// TIA Portal V19 export
ORGANIZATION_BLOCK "Main_hw"   // OB124, LAD, ProgramCycle
TITLE = "Main Program Sweep (Cycle)"
{ S7_Optimized_Access := 'TRUE' }
// stored: SetENOAutomatically false
   VAR_INPUT
      Initial_Call : Bool;   // Initial call of this OB
      Remanence : Bool;   // =True, if remanent data are available
   END_VAR
   VAR_TEMP   // added for the SCL form of the ladder/FBD networks
      _w1 : Bool;
      _w2 : Bool;
   END_VAR
BEGIN

REGION Network 1: HMI hardware test screen control
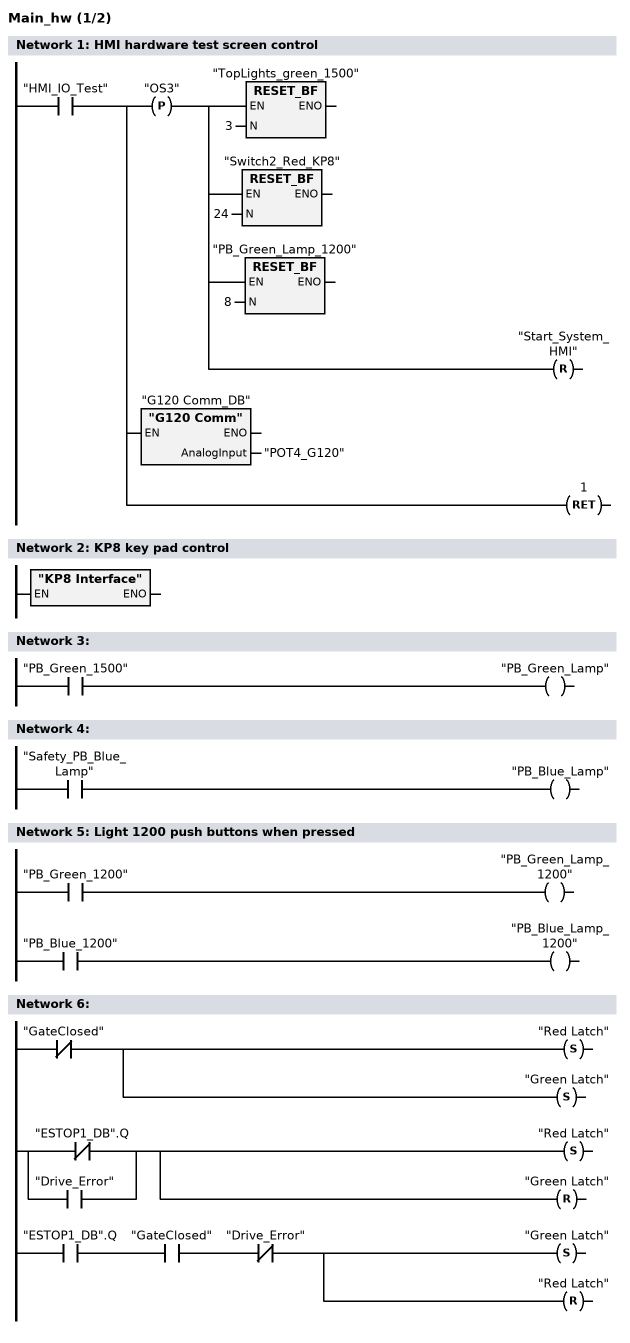
   // no SCL statement known for RBitfield: written as a call
   #_w1 := "HMI_IO_Test" AND NOT "OS3";   // rising edge
   "OS3" := "HMI_IO_Test";
   #_w2 := "HMI_IO_Test";
   IF #_w1 THEN
       RESET_BF(operand := "TopLights_green_1500", n := 3);
       RESET_BF(operand := "Switch2_Red_KP8", n := 24);
       RESET_BF(operand := "PB_Green_Lamp_1200", n := 8);
       "Start_System_HMI" := FALSE;
   END_IF;
   IF #_w2 THEN
       "G120 Comm_DB"(AnalogInput => "POT4_G120");   // "G120 Comm"
       ENO := 1;
       RETURN;
   END_IF;
END_REGION

REGION Network 2: KP8 key pad control
   RUNG wire#powerrail
      "KP8 Interface"()
   END_RUNG
   // the same network as SCL:
   "KP8 Interface"();
END_REGION

REGION Network 3
   RUNG wire#powerrail
      Contact( "PB_Green_1500" )
      Coil( "PB_Green_Lamp" )
   END_RUNG
   // the same network as SCL:
   "PB_Green_Lamp" := "PB_Green_1500";
END_REGION

REGION Network 4
   RUNG wire#powerrail
      Contact( "Safety_PB_Blue_Lamp" )
      Coil( "PB_Blue_Lamp" )
   END_RUNG
   // the same network as SCL:
   "PB_Blue_Lamp" := "Safety_PB_Blue_Lamp";
END_REGION

REGION Network 5: Light 1200 push buttons when pressed
   RUNG wire#powerrail
      Contact( "PB_Green_1200" )
      Coil( "PB_Green_Lamp_1200" )
   END_RUNG
   RUNG wire#powerrail
      Contact( "PB_Blue_1200" )
      Coil( "PB_Blue_Lamp_1200" )
   END_RUNG
   // the same network as SCL:
   "PB_Green_Lamp_1200" := "PB_Green_1200";
   "PB_Blue_Lamp_1200" := "PB_Blue_1200";
END_REGION

REGION Network 6
   RUNG wire#powerrail
      I_Contact( "GateClosed" )
      wire#w1
      S_Coil( "Red Latch" )
   END_RUNG
   RUNG wire#w1
      S_Coil( "Green Latch" )
   END_RUNG
   RUNG wire#powerrail
      I_Contact( "ESTOP1_DB".Q )
      wire#w2
      S_Coil( "Red Latch" )
   END_RUNG
   RUNG wire#powerrail
      Contact( "Drive_Error" )
   END_RUNG wire#w2
   RUNG wire#w2
      R_Coil( "Green Latch" )
   END_RUNG
   RUNG wire#powerrail
      Contact( "ESTOP1_DB".Q )
      Contact( "GateClosed" )
      I_Contact( "Drive_Error" )
      wire#w3
      S_Coil( "Green Latch" )
   END_RUNG
   RUNG wire#w3
      R_Coil( "Red Latch" )
   END_RUNG
   // the same network as SCL:
   IF NOT "GateClosed" THEN
       "Red Latch" := TRUE;
       "Green Latch" := TRUE;
   END_IF;
   IF NOT "ESTOP1_DB".Q OR "Drive_Error" THEN
       "Red Latch" := TRUE;
       "Green Latch" := FALSE;
   END_IF;
   IF "ESTOP1_DB".Q AND "GateClosed" AND NOT "Drive_Error" THEN
       "Green Latch" := TRUE;
       "Red Latch" := FALSE;
   END_IF;
END_REGION

REGION Network 7
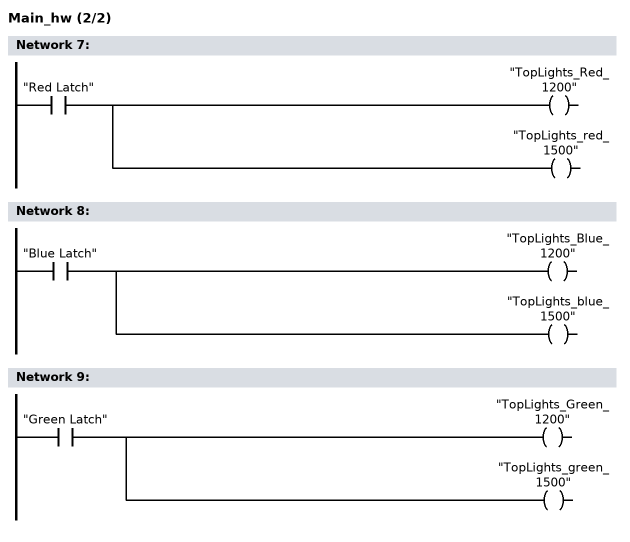
   RUNG wire#powerrail
      Contact( "Red Latch" )
      wire#w1
      Coil( "TopLights_Red_1200" )
   END_RUNG
   RUNG wire#w1
      Coil( "TopLights_red_1500" )
   END_RUNG
   // the same network as SCL:
   "TopLights_Red_1200" := "Red Latch";
   "TopLights_red_1500" := "Red Latch";
END_REGION

REGION Network 8
   RUNG wire#powerrail
      Contact( "Blue Latch" )
      wire#w1
      Coil( "TopLights_Blue_1200" )
   END_RUNG
   RUNG wire#w1
      Coil( "TopLights_blue_1500" )
   END_RUNG
   // the same network as SCL:
   "TopLights_Blue_1200" := "Blue Latch";
   "TopLights_blue_1500" := "Blue Latch";
END_REGION

REGION Network 9
   RUNG wire#powerrail
      Contact( "Green Latch" )
      wire#w1
      Coil( "TopLights_Green_1200" )
   END_RUNG
   RUNG wire#w1
      Coil( "TopLights_green_1500" )
   END_RUNG
   // the same network as SCL:
   "TopLights_Green_1200" := "Green Latch";
   "TopLights_green_1500" := "Green Latch";
END_REGION
END_ORGANIZATION_BLOCK
